TEXTLIST WorkAreaStatePN
  0 = 'Positive'
  1 = 'Negative'
   = ''
END_TEXTLIST

(* stored: Version 1.1.0.1, ProductVersion 3.1.4024.11
   TextList WorkAreaStatePN: Id {b58e5be8-2caf-4c31-bcae-165c9f404e72} *)
